{attribute addProperty BoxType "EL6690-0002-0000"}
{attribute addProperty Id "StatusAT %I*Status_93A34D63810InputsEMPTY_STRUCTURE000OutputsEMPTY_STRUCTURE000WcStateAT %I*WcState_F855686C1620InfoDataAT %I*InfoData_192954DE1620"}
{attribute addProperty CRC "3145171794"}
{attribute addProperty SizeInBites "40"}
{attribute addProperty SizeInBytes "5"}
TYPE EL6690_04D299B4 :
STRUCT
	{attribute addProperty Name "Status"}
	Status : Status_93A34D63;
	{attribute addProperty Name "Inputs"}
	Inputs : EMPTY_STRUCTURE;
	{attribute addProperty Name "Outputs"}
	Outputs : EMPTY_STRUCTURE;
	{attribute addProperty Name "WcState"}
	WcState : WcState_F855686C;
	{attribute addProperty Name "InfoData"}
	InfoData : InfoData_192954DE;
END_STRUCT
END_TYPE

(* stored: Version 1.2.0.0, ProductVersion 3.1.4024.9
   DUT EL6690_04D299B4: Id {9a1e45fe-bc95-4676-9b93-bb11373d6556} *)
